INTERFACE I_Testsuite EXTENDS I_Base

PROPERTY PUBLIC P_Assertions : int
GET
END_GET
END_PROPERTY

PROPERTY PUBLIC P_Errors : int
GET
END_GET
END_PROPERTY

PROPERTY PUBLIC P_Failures : int
GET
END_GET
END_PROPERTY

PROPERTY PUBLIC P_File : STRING(255)
GET
END_GET
SET
END_SET
END_PROPERTY

PROPERTY PUBLIC P_Skipped : int
GET
END_GET
END_PROPERTY

PROPERTY PUBLIC P_Tests : int
GET
END_GET
END_PROPERTY

PROPERTY PUBLIC P_Time : LREAL
GET
END_GET
SET
END_SET
END_PROPERTY

PROPERTY PUBLIC P_Timestamp : String(39)
GET
END_GET
SET
END_SET
END_PROPERTY

END_INTERFACE

(* stored: Version 1.1.0.1
   Itf I_Testsuite: Id {be1b8503-88c7-00d0-316f-5b2753f7b610}
   Property P_Assertions: Id {592ea10d-e304-0be1-2ca9-b718e1bb8709}
   Get Get: Id {167fc972-868f-07ff-0df6-5c8fbbafb0ec}
   Property P_Errors: Id {d81823f9-f404-01b7-05bf-8e15a401d543}
   Get Get: Id {66593c04-dc5d-025c-2e4b-d15d0cd4d037}
   Property P_Failures: Id {917df731-91c8-009f-256a-584de2d1943f}
   Get Get: Id {13e47927-db5e-0662-033a-00390df5b562}
   Property P_File: Id {bb667d1a-7641-01af-115e-dad5d58eeeb6}
   Get Get: Id {0987e319-b31e-02d0-11f9-c85c651a4a3a}
   Set Set: Id {8d03ead8-bfec-0c00-3960-89537ab0d853}
   Property P_Skipped: Id {39fbdb3e-86fe-0711-31f2-83215633aa4f}
   Get Get: Id {30715938-b42c-02a4-25f6-1f41efc18665}
   Property P_Tests: Id {39a38ba9-e262-08af-172f-beb45ec34a85}
   Get Get: Id {215f9cb0-0610-001b-059c-7a303c71b9aa}
   Property P_Time: Id {c6aa324d-dcec-0fb7-29ce-a6a764884bdf}
   Get Get: Id {724e0ce4-d387-0861-0358-a63e1bba51c3}
   Set Set: Id {3208e591-5717-0959-1457-8475838628e3}
   Property P_Timestamp: Id {88083642-b2c3-0152-1ed9-0e2fb12145fd}
   Get Get: Id {1f62dac4-2539-0718-378b-6b2a098b196c}
   Set Set: Id {56bdb73c-92ec-0add-0b26-48a44ae6f8ee} *)
